ABB RAPID module: Module1.mod

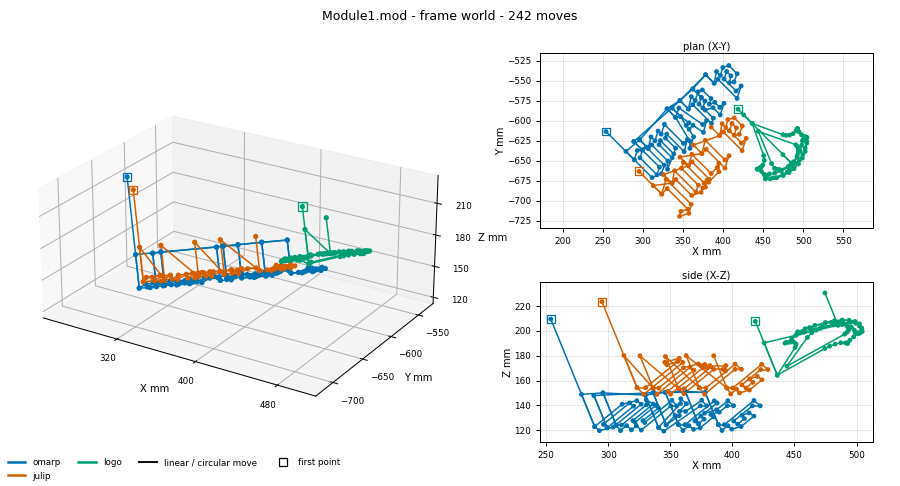
[picture p0: tool path of Module1.mod in frame world, 242 of 244 moves have a stored position in this frame; points joined in program order, loops and branches not executed]
MODULE Module1
    PERS tooldata toolx:=[TRUE,[[148.954,0,67.083],[0.79335334,0,0.608761429,0]],[1,[0,0,1],[1,0,0,0],0,0,0]];
    TASK PERS wobjdata Workobject_2:=[FALSE,TRUE,"",[[233.257625,-636.839625,95.228693814],[0.892399134,-0.099045186,-0.239118017,-0.369643626]],[[0,0,0],[1,0,0,0]]];
    CONST robtarget Target_10:=[[55.302,30.991,100],[0,0,1,0],[-1,1,-2,0],[9E+09,9E+09,9E+09,9E+09,9E+09,9E+09]];
    CONST robtarget Target_20:=[[55.302,30.991,0],[0,0,1,0],[-1,1,-2,0],[9E+09,9E+09,9E+09,9E+09,9E+09,9E+09]];
    CONST robtarget Target_30:=[[91.365,30.991,0],[0,0,1,0],[-1,1,-2,0],[9E+09,9E+09,9E+09,9E+09,9E+09,9E+09]];
    CONST robtarget Target_40:=[[97.105,42.767,0],[0,0,1,0],[-1,1,-2,0],[9E+09,9E+09,9E+09,9E+09,9E+09,9E+09]];
    CONST robtarget Target_50:=[[91.365,52.776,0],[0,0,1,0],[-1,1,-2,0],[9E+09,9E+09,9E+09,9E+09,9E+09,9E+09]];
    CONST robtarget Target_60:=[[54.418,52.776,0],[0,0,1,0],[-1,1,-2,0],[9E+09,9E+09,9E+09,9E+09,9E+09,9E+09]];
    CONST robtarget Target_70:=[[48.825,41.884,0],[0,0,1,0],[-1,1,-2,0],[9E+09,9E+09,9E+09,9E+09,9E+09,9E+09]];
    CONST robtarget Target_80:=[[55.302,30.991,0],[0,0,1,0],[-1,1,-2,0],[9E+09,9E+09,9E+09,9E+09,9E+09,9E+09]];
    CONST robtarget Target_90:=[[55.302,30.991,30],[0,0,1,0],[-1,1,-2,0],[9E+09,9E+09,9E+09,9E+09,9E+09,9E+09]];
    CONST robtarget Target_100:=[[57.714,53.347,30],[0,0,1,0],[-1,1,-2,0],[9E+09,9E+09,9E+09,9E+09,9E+09,9E+09]];
    CONST robtarget Target_110:=[[57.714,53.347,0],[0,0,1,0],[-1,1,-2,0],[9E+09,9E+09,9E+09,9E+09,9E+09,9E+09]];
    CONST robtarget Target_120:=[[57.714,59.499,0],[0,0,1,0],[-1,1,-2,0],[9E+09,9E+09,9E+09,9E+09,9E+09,9E+09]];
    CONST robtarget Target_130:=[[90.706,59.499,0],[0,0,1,0],[-1,1,-2,0],[9E+09,9E+09,9E+09,9E+09,9E+09,9E+09]];
    CONST robtarget Target_140:=[[98.758,51.972,0],[0,0,1,0],[-1,1,-2,0],[9E+09,9E+09,9E+09,9E+09,9E+09,9E+09]];
    CONST robtarget Target_150:=[[91.756,66.151,0],[0,0,1,0],[-1,1,-2,0],[9E+09,9E+09,9E+09,9E+09,9E+09,9E+09]];
    CONST robtarget Target_160:=[[64.974,66.151,0],[0,0,1,0],[-1,1,-2,0],[9E+09,9E+09,9E+09,9E+09,9E+09,9E+09]];
    CONST robtarget Target_170:=[[62.173,71.052,0],[0,0,1,0],[-1,1,-2,0],[9E+09,9E+09,9E+09,9E+09,9E+09,9E+09]];
    CONST robtarget Target_180:=[[89.48,71.052,0],[0,0,1,0],[-1,1,-2,0],[9E+09,9E+09,9E+09,9E+09,9E+09,9E+09]];
    CONST robtarget Target_190:=[[85.36,77.652,0],[0,0,1,0],[-1,1,-2,0],[9E+09,9E+09,9E+09,9E+09,9E+09,9E+09]];
    CONST robtarget Target_200:=[[64.9,77.652,0],[0,0,1,0],[-1,1,-2,0],[9E+09,9E+09,9E+09,9E+09,9E+09,9E+09]];
    CONST robtarget Target_210:=[[61.956,82.215,0],[0,0,1,0],[-1,1,-2,0],[9E+09,9E+09,9E+09,9E+09,9E+09,9E+09]];
    CONST robtarget Target_220:=[[97.748,82.215,0],[0,0,1,0],[-1,1,-2,0],[9E+09,9E+09,9E+09,9E+09,9E+09,9E+09]];
    CONST robtarget Target_230:=[[88.605,95.734,0],[0,0,1,0],[-1,1,-2,0],[9E+09,9E+09,9E+09,9E+09,9E+09,9E+09]];
    CONST robtarget Target_240:=[[88.605,88.907,0],[0,0,1,0],[-1,1,-2,0],[9E+09,9E+09,9E+09,9E+09,9E+09,9E+09]];
    CONST robtarget Target_250:=[[49.745,88.907,0],[0,0,1,0],[-1,1,-2,0],[9E+09,9E+09,9E+09,9E+09,9E+09,9E+09]];
    CONST robtarget Target_260:=[[56.572,77.354,0],[0,0,1,0],[-1,1,-2,0],[9E+09,9E+09,9E+09,9E+09,9E+09,9E+09]];
    CONST robtarget Target_270:=[[50.095,77.354,0],[0,0,1,0],[-1,1,-2,0],[9E+09,9E+09,9E+09,9E+09,9E+09,9E+09]];
    CONST robtarget Target_280:=[[56.922,65.976,0],[0,0,1,0],[-1,1,-2,0],[9E+09,9E+09,9E+09,9E+09,9E+09,9E+09]];
    CONST robtarget Target_290:=[[48.87,65.976,0],[0,0,1,0],[-1,1,-2,0],[9E+09,9E+09,9E+09,9E+09,9E+09,9E+09]];
    CONST robtarget Target_300:=[[57.714,53.347,0],[0,0,1,0],[-1,1,-2,0],[9E+09,9E+09,9E+09,9E+09,9E+09,9E+09]];
    CONST robtarget Target_310:=[[57.714,53.347,30],[0,0,1,0],[-1,1,-2,0],[9E+09,9E+09,9E+09,9E+09,9E+09,9E+09]];
    CONST robtarget Target_320:=[[53.98,104.878,30],[0,0,1,0],[-1,1,-2,0],[9E+09,9E+09,9E+09,9E+09,9E+09,9E+09]];
    CONST robtarget Target_330:=[[53.98,104.878,0],[0,0,1,0],[-1,1,-2,0],[9E+09,9E+09,9E+09,9E+09,9E+09,9E+09]];
    CONST robtarget Target_340:=[[92.492,96.56,0],[0,0,1,0],[-1,1,-2,0],[9E+09,9E+09,9E+09,9E+09,9E+09,9E+09]];
    CONST robtarget Target_350:=[[100.22,90.23,0],[0,0,1,0],[-1,1,-2,0],[9E+09,9E+09,9E+09,9E+09,9E+09,9E+09]];
    CONST robtarget Target_360:=[[92.179,103.629,0],[0,0,1,0],[-1,1,-2,0],[9E+09,9E+09,9E+09,9E+09,9E+09,9E+09]];
    CONST robtarget Target_370:=[[79.793,106.336,0],[0,0,1,0],[-1,1,-2,0],[9E+09,9E+09,9E+09,9E+09,9E+09,9E+09]];
    CONST robtarget Target_380:=[[79.793,113.309,0],[0,0,1,0],[-1,1,-2,0],[9E+09,9E+09,9E+09,9E+09,9E+09,9E+09]];
    CONST robtarget Target_390:=[[97.695,116.224,0],[0,0,1,0],[-1,1,-2,0],[9E+09,9E+09,9E+09,9E+09,9E+09,9E+09]];
    CONST robtarget Target_400:=[[88.848,129.546,0],[0,0,1,0],[-1,1,-2,0],[9E+09,9E+09,9E+09,9E+09,9E+09,9E+09]];
    CONST robtarget Target_410:=[[88.848,122.469,0],[0,0,1,0],[-1,1,-2,0],[9E+09,9E+09,9E+09,9E+09,9E+09,9E+09]];
    CONST robtarget Target_420:=[[47.943,116.119,0],[0,0,1,0],[-1,1,-2,0],[9E+09,9E+09,9E+09,9E+09,9E+09,9E+09]];
    CONST robtarget Target_430:=[[53.98,104.878,0],[0,0,1,0],[-1,1,-2,0],[9E+09,9E+09,9E+09,9E+09,9E+09,9E+09]];
    CONST robtarget Target_440:=[[53.98,104.878,30],[0,0,1,0],[-1,1,-2,0],[9E+09,9E+09,9E+09,9E+09,9E+09,9E+09]];
    CONST robtarget Target_450:=[[58.556,123.595,30],[0,0,1,0],[-1,1,-2,0],[9E+09,9E+09,9E+09,9E+09,9E+09,9E+09]];
    CONST robtarget Target_460:=[[58.556,123.595,0],[0,0,1,0],[-1,1,-2,0],[9E+09,9E+09,9E+09,9E+09,9E+09,9E+09]];
    CONST robtarget Target_470:=[[58.556,131.263,0],[0,0,1,0],[-1,1,-2,0],[9E+09,9E+09,9E+09,9E+09,9E+09,9E+09]];
    CONST robtarget Target_480:=[[96.839,131.263,0],[0,0,1,0],[-1,1,-2,0],[9E+09,9E+09,9E+09,9E+09,9E+09,9E+09]];
    CONST robtarget Target_490:=[[93.38,137.518,0],[0,0,1,0],[-1,1,-2,0],[9E+09,9E+09,9E+09,9E+09,9E+09,9E+09]];
    CONST robtarget Target_500:=[[76.894,137.518,0],[0,0,1,0],[-1,1,-2,0],[9E+09,9E+09,9E+09,9E+09,9E+09,9E+09]];
    CONST robtarget Target_510:=[[82.34,146.497,0],[0,0,1,0],[-1,1,-2,0],[9E+09,9E+09,9E+09,9E+09,9E+09,9E+09]];
    CONST robtarget Target_520:=[[97.06,146.497,0],[0,0,1,0],[-1,1,-2,0],[9E+09,9E+09,9E+09,9E+09,9E+09,9E+09]];
    CONST robtarget Target_530:=[[89.004,160.012,0],[0,0,1,0],[-1,1,-2,0],[9E+09,9E+09,9E+09,9E+09,9E+09,9E+09]];
    CONST robtarget Target_540:=[[89.004,152.806,0],[0,0,1,0],[-1,1,-2,0],[9E+09,9E+09,9E+09,9E+09,9E+09,9E+09]];
    CONST robtarget Target_550:=[[78.627,152.806,0],[0,0,1,0],[-1,1,-2,0],[9E+09,9E+09,9E+09,9E+09,9E+09,9E+09]];
    CONST robtarget Target_560:=[[75.018,146.246,0],[0,0,1,0],[-1,1,-2,0],[9E+09,9E+09,9E+09,9E+09,9E+09,9E+09]];
    CONST robtarget Target_570:=[[71.057,152.806,0],[0,0,1,0],[-1,1,-2,0],[9E+09,9E+09,9E+09,9E+09,9E+09,9E+09]];
    CONST robtarget Target_580:=[[53.357,152.806,0],[0,0,1,0],[-1,1,-2,0],[9E+09,9E+09,9E+09,9E+09,9E+09,9E+09]];
    CONST robtarget Target_590:=[[50.882,147.483,0],[0,0,1,0],[-1,1,-2,0],[9E+09,9E+09,9E+09,9E+09,9E+09,9E+09]];
    CONST robtarget Target_600:=[[56.823,137.086,0],[0,0,1,0],[-1,1,-2,0],[9E+09,9E+09,9E+09,9E+09,9E+09,9E+09]];
    CONST robtarget Target_610:=[[48.901,137.086,0],[0,0,1,0],[-1,1,-2,0],[9E+09,9E+09,9E+09,9E+09,9E+09,9E+09]];
    CONST robtarget Target_620:=[[58.556,123.595,0],[0,0,1,0],[-1,1,-2,0],[9E+09,9E+09,9E+09,9E+09,9E+09,9E+09]];
    CONST robtarget Target_630:=[[58.556,123.595,30],[0,0,1,0],[-1,1,-2,0],[9E+09,9E+09,9E+09,9E+09,9E+09,9E+09]];
    CONST robtarget Target_640:=[[58.524,169.09,30],[0,0,1,0],[-1,1,-2,0],[9E+09,9E+09,9E+09,9E+09,9E+09,9E+09]];
    CONST robtarget Target_650:=[[58.524,169.09,0],[0,0,1,0],[-1,1,-2,0],[9E+09,9E+09,9E+09,9E+09,9E+09,9E+09]];
    CONST robtarget Target_660:=[[58.524,175.96,0],[0,0,1,0],[-1,1,-2,0],[9E+09,9E+09,9E+09,9E+09,9E+09,9E+09]];
    CONST robtarget Target_670:=[[97.451,175.96,0],[0,0,1,0],[-1,1,-2,0],[9E+09,9E+09,9E+09,9E+09,9E+09,9E+09]];
    CONST robtarget Target_680:=[[88.812,190.531,0],[0,0,1,0],[-1,1,-2,0],[9E+09,9E+09,9E+09,9E+09,9E+09,9E+09]];
    CONST robtarget Target_690:=[[88.812,181.58,0],[0,0,1,0],[-1,1,-2,0],[9E+09,9E+09,9E+09,9E+09,9E+09,9E+09]];
    CONST robtarget Target_700:=[[64.353,181.58,0],[0,0,1,0],[-1,1,-2,0],[9E+09,9E+09,9E+09,9E+09,9E+09,9E+09]];
    CONST robtarget Target_710:=[[59.253,190.427,0],[0,0,1,0],[-1,1,-2,0],[9E+09,9E+09,9E+09,9E+09,9E+09,9E+09]];
    CONST robtarget Target_720:=[[68.204,190.427,0],[0,0,1,0],[-1,1,-2,0],[9E+09,9E+09,9E+09,9E+09,9E+09,9E+09]];
    CONST robtarget Target_730:=[[73.512,182.933,0],[0,0,1,0],[-1,1,-2,0],[9E+09,9E+09,9E+09,9E+09,9E+09,9E+09]];
    CONST robtarget Target_740:=[[77.467,187.721,0],[0,0,1,0],[-1,1,-2,0],[9E+09,9E+09,9E+09,9E+09,9E+09,9E+09]];
    CONST robtarget Target_750:=[[72.263,197.713,0],[0,0,1,0],[-1,1,-2,0],[9E+09,9E+09,9E+09,9E+09,9E+09,9E+09]];
    CONST robtarget Target_760:=[[55.506,197.713,0],[0,0,1,0],[-1,1,-2,0],[9E+09,9E+09,9E+09,9E+09,9E+09,9E+09]];
    CONST robtarget Target_770:=[[51.238,190.635,0],[0,0,1,0],[-1,1,-2,0],[9E+09,9E+09,9E+09,9E+09,9E+09,9E+09]];
    CONST robtarget Target_780:=[[56.859,181.476,0],[0,0,1,0],[-1,1,-2,0],[9E+09,9E+09,9E+09,9E+09,9E+09,9E+09]];
    CONST robtarget Target_790:=[[49.053,181.476,0],[0,0,1,0],[-1,1,-2,0],[9E+09,9E+09,9E+09,9E+09,9E+09,9E+09]];
    CONST robtarget Target_800:=[[58.524,169.09,0],[0,0,1,0],[-1,1,-2,0],[9E+09,9E+09,9E+09,9E+09,9E+09,9E+09]];
    CONST robtarget Target_810:=[[58.524,169.09,30],[0,0,1,0],[-1,1,-2,0],[9E+09,9E+09,9E+09,9E+09,9E+09,9E+09]];
    CONST robtarget Target_820:=[[59.96,145.179,30],[0,0,1,0],[-1,1,-2,0],[9E+09,9E+09,9E+09,9E+09,9E+09,9E+09]];
    CONST robtarget Target_830:=[[59.96,145.179,0],[0,0,1,0],[-1,1,-2,0],[9E+09,9E+09,9E+09,9E+09,9E+09,9E+09]];
    CONST robtarget Target_840:=[[64.416,137.257,0],[0,0,1,0],[-1,1,-2,0],[9E+09,9E+09,9E+09,9E+09,9E+09,9E+09]];
    CONST robtarget Target_850:=[[72.461,137.257,0],[0,0,1,0],[-1,1,-2,0],[9E+09,9E+09,9E+09,9E+09,9E+09,9E+09]];
    CONST robtarget Target_860:=[[67.386,145.179,0],[0,0,1,0],[-1,1,-2,0],[9E+09,9E+09,9E+09,9E+09,9E+09,9E+09]];
    CONST robtarget Target_870:=[[59.96,145.179,0],[0,0,1,0],[-1,1,-2,0],[9E+09,9E+09,9E+09,9E+09,9E+09,9E+09]];
    CONST robtarget Target_880:=[[59.96,145.179,30],[0,0,1,0],[-1,1,-2,0],[9E+09,9E+09,9E+09,9E+09,9E+09,9E+09]];
    CONST robtarget Target_890:=[[58.039,110.083,30],[0,0,1,0],[-1,1,-2,0],[9E+09,9E+09,9E+09,9E+09,9E+09,9E+09]];
    CONST robtarget Target_900:=[[58.039,110.083,0],[0,0,1,0],[-1,1,-2,0],[9E+09,9E+09,9E+09,9E+09,9E+09,9E+09]];
    CONST robtarget Target_910:=[[73.132,107.168,0],[0,0,1,0],[-1,1,-2,0],[9E+09,9E+09,9E+09,9E+09,9E+09,9E+09]];
    CONST robtarget Target_920:=[[73.132,111.956,0],[0,0,1,0],[-1,1,-2,0],[9E+09,9E+09,9E+09,9E+09,9E+09,9E+09]];
    CONST robtarget Target_930:=[[58.039,110.083,0],[0,0,1,0],[-1,1,-2,0],[9E+09,9E+09,9E+09,9E+09,9E+09,9E+09]];
    CONST robtarget Target_940:=[[58.039,110.083,30],[0,0,1,0],[-1,1,-2,0],[9E+09,9E+09,9E+09,9E+09,9E+09,9E+09]];
    CONST robtarget Target_950:=[[53.478,46.741,30],[0,0,1,0],[-1,1,-2,0],[9E+09,9E+09,9E+09,9E+09,9E+09,9E+09]];
    CONST robtarget Target_960:=[[53.478,46.741,0],[0,0,1,0],[-1,1,-2,0],[9E+09,9E+09,9E+09,9E+09,9E+09,9E+09]];
    CONST robtarget Target_970:=[[58.982,37.762,0],[0,0,1,0],[-1,1,-2,0],[9E+09,9E+09,9E+09,9E+09,9E+09,9E+09]];
    CONST robtarget Target_980:=[[93.58,37.762,0],[0,0,1,0],[-1,1,-2,0],[9E+09,9E+09,9E+09,9E+09,9E+09,9E+09]];
    CONST robtarget Target_990:=[[88.274,46.741,0],[0,0,1,0],[-1,1,-2,0],[9E+09,9E+09,9E+09,9E+09,9E+09,9E+09]];
    CONST robtarget Target_1000:=[[53.478,46.741,0],[0,0,1,0],[-1,1,-2,0],[9E+09,9E+09,9E+09,9E+09,9E+09,9E+09]];
    CONST robtarget Target_1010:=[[53.478,46.741,30],[0,0,1,0],[-1,1,-2,0],[9E+09,9E+09,9E+09,9E+09,9E+09,9E+09]];
    CONST jointtarget JointTarget_3:=[[0,0,0,0,0,0],[9E+09,9E+09,9E+09,9E+09,9E+09,9E+09]];
    CONST robtarget Target_1020:=[[118.053795712,24.917790512,80],[0,0,1,0],[-1,1,-2,0],[9E+09,9E+09,9E+09,9E+09,9E+09,9E+09]];
    CONST robtarget Target_1030:=[[118.054,24.918,0],[0,0,1,0],[-1,1,-2,0],[9E+09,9E+09,9E+09,9E+09,9E+09,9E+09]];
    CONST robtarget Target_1040:=[[118.054,34.711,0],[0,0,1,0],[-1,1,-2,0],[9E+09,9E+09,9E+09,9E+09,9E+09,9E+09]];
    CONST robtarget Target_1050:=[[160.24,34.711,0],[0,0,1,0],[-1,1,-2,0],[9E+09,9E+09,9E+09,9E+09,9E+09,9E+09]];
    CONST robtarget Target_1060:=[[155.164,26.659,0],[0,0,1,0],[-1,1,-2,0],[9E+09,9E+09,9E+09,9E+09,9E+09,9E+09]];
    CONST robtarget Target_1070:=[[159.015,21.058,0],[0,0,1,0],[-1,1,-2,0],[9E+09,9E+09,9E+09,9E+09,9E+09,9E+09]];
    CONST robtarget Target_1080:=[[165.492,31.911,0],[0,0,1,0],[-1,1,-2,0],[9E+09,9E+09,9E+09,9E+09,9E+09,9E+09]];
    CONST robtarget Target_1090:=[[158.665,41.888,0],[0,0,1,0],[-1,1,-2,0],[9E+09,9E+09,9E+09,9E+09,9E+09,9E+09]];
    CONST robtarget Target_1100:=[[107.376,41.888,0],[0,0,1,0],[-1,1,-2,0],[9E+09,9E+09,9E+09,9E+09,9E+09,9E+09]];
    CONST robtarget Target_1110:=[[118.054,24.918,0],[0,0,1,0],[-1,1,-2,0],[9E+09,9E+09,9E+09,9E+09,9E+09,9E+09]];
    CONST robtarget Target_1120:=[[118.054,24.918,30],[0,0,1,0],[-1,1,-2,0],[9E+09,9E+09,9E+09,9E+09,9E+09,9E+09]];
    CONST robtarget Target_1130:=[[117.489,43.728,0],[0,0,1,0],[-1,1,-2,0],[9E+09,9E+09,9E+09,9E+09,9E+09,9E+09]];
    CONST robtarget Target_1140:=[[117.489,50.177,0],[0,0,1,0],[-1,1,-2,0],[9E+09,9E+09,9E+09,9E+09,9E+09,9E+09]];
    CONST robtarget Target_1150:=[[150.072,50.177,0],[0,0,1,0],[-1,1,-2,0],[9E+09,9E+09,9E+09,9E+09,9E+09,9E+09]];
    CONST robtarget Target_1160:=[[156.421,61.314,0],[0,0,1,0],[-1,1,-2,0],[9E+09,9E+09,9E+09,9E+09,9E+09,9E+09]];
    CONST robtarget Target_1170:=[[153.61,66.726,0],[0,0,1,0],[-1,1,-2,0],[9E+09,9E+09,9E+09,9E+09,9E+09,9E+09]];
    CONST robtarget Target_1180:=[[155.588,69.745,0],[0,0,1,0],[-1,1,-2,0],[9E+09,9E+09,9E+09,9E+09,9E+09,9E+09]];
    CONST robtarget Target_1190:=[[150.072,77.343,0],[0,0,1,0],[-1,1,-2,0],[9E+09,9E+09,9E+09,9E+09,9E+09,9E+09]];
    CONST robtarget Target_1200:=[[150.072,72.176,0],[0,0,1,0],[-1,1,-2,0],[9E+09,9E+09,9E+09,9E+09,9E+09,9E+09]];
    CONST robtarget Target_1210:=[[107.603,72.176,0],[0,0,1,0],[-1,1,-2,0],[9E+09,9E+09,9E+09,9E+09,9E+09,9E+09]];
    CONST robtarget Target_1220:=[[111.979,65.13,0],[0,0,1,0],[-1,1,-2,0],[9E+09,9E+09,9E+09,9E+09,9E+09,9E+09]];
    CONST robtarget Target_1230:=[[146.392,65.13,0],[0,0,1,0],[-1,1,-2,0],[9E+09,9E+09,9E+09,9E+09,9E+09,9E+09]];
    CONST robtarget Target_1240:=[[150.91,56.876,0],[0,0,1,0],[-1,1,-2,0],[9E+09,9E+09,9E+09,9E+09,9E+09,9E+09]];
    CONST robtarget Target_1250:=[[107.381,56.876,0],[0,0,1,0],[-1,1,-2,0],[9E+09,9E+09,9E+09,9E+09,9E+09,9E+09]];
    CONST robtarget Target_1260:=[[117.489,43.728,0],[0,0,1,0],[-1,1,-2,0],[9E+09,9E+09,9E+09,9E+09,9E+09,9E+09]];
    CONST robtarget Target_1270:=[[117.489,43.728,30],[0,0,1,0],[-1,1,-2,0],[9E+09,9E+09,9E+09,9E+09,9E+09,9E+09]];
    CONST robtarget Target_1280:=[[116.365,73.7,0],[0,0,1,0],[-1,1,-2,0],[9E+09,9E+09,9E+09,9E+09,9E+09,9E+09]];
    CONST robtarget Target_1290:=[[116.365,80.093,0],[0,0,1,0],[-1,1,-2,0],[9E+09,9E+09,9E+09,9E+09,9E+09,9E+09]];
    CONST robtarget Target_1300:=[[151.605,80.093,0],[0,0,1,0],[-1,1,-2,0],[9E+09,9E+09,9E+09,9E+09,9E+09,9E+09]];
    CONST robtarget Target_1310:=[[153.709,76.813,0],[0,0,1,0],[-1,1,-2,0],[9E+09,9E+09,9E+09,9E+09,9E+09,9E+09]];
    CONST robtarget Target_1320:=[[153.709,95.194,0],[0,0,1,0],[-1,1,-2,0],[9E+09,9E+09,9E+09,9E+09,9E+09,9E+09]];
    CONST robtarget Target_1330:=[[144.921,102.496,0],[0,0,1,0],[-1,1,-2,0],[9E+09,9E+09,9E+09,9E+09,9E+09,9E+09]];
    CONST robtarget Target_1340:=[[147.621,97.284,0],[0,0,1,0],[-1,1,-2,0],[9E+09,9E+09,9E+09,9E+09,9E+09,9E+09]];
    CONST robtarget Target_1350:=[[147.621,86.727,0],[0,0,1,0],[-1,1,-2,0],[9E+09,9E+09,9E+09,9E+09,9E+09,9E+09]];
    CONST robtarget Target_1360:=[[108.343,86.727,0],[0,0,1,0],[-1,1,-2,0],[9E+09,9E+09,9E+09,9E+09,9E+09,9E+09]];
    CONST robtarget Target_1370:=[[116.365,73.7,0],[0,0,1,0],[-1,1,-2,0],[9E+09,9E+09,9E+09,9E+09,9E+09,9E+09]];
    CONST robtarget Target_1380:=[[116.365,73.7,30],[0,0,1,0],[-1,1,-2,0],[9E+09,9E+09,9E+09,9E+09,9E+09,9E+09]];
    CONST robtarget Target_1390:=[[117.776,96.145,0],[0,0,1,0],[-1,1,-2,0],[9E+09,9E+09,9E+09,9E+09,9E+09,9E+09]];
    CONST robtarget Target_1400:=[[117.776,103.695,0],[0,0,1,0],[-1,1,-2,0],[9E+09,9E+09,9E+09,9E+09,9E+09,9E+09]];
    CONST robtarget Target_1410:=[[156.047,103.695,0],[0,0,1,0],[-1,1,-2,0],[9E+09,9E+09,9E+09,9E+09,9E+09,9E+09]];
    CONST robtarget Target_1420:=[[147.621,118.268,0],[0,0,1,0],[-1,1,-2,0],[9E+09,9E+09,9E+09,9E+09,9E+09,9E+09]];
    CONST robtarget Target_1430:=[[147.621,110.908,0],[0,0,1,0],[-1,1,-2,0],[9E+09,9E+09,9E+09,9E+09,9E+09,9E+09]];
    CONST robtarget Target_1440:=[[107.62,110.908,0],[0,0,1,0],[-1,1,-2,0],[9E+09,9E+09,9E+09,9E+09,9E+09,9E+09]];
    CONST robtarget Target_1450:=[[117.776,96.145,0],[0,0,1,0],[-1,1,-2,0],[9E+09,9E+09,9E+09,9E+09,9E+09,9E+09]];
    CONST robtarget Target_1460:=[[117.776,96.145,30],[0,0,1,0],[-1,1,-2,0],[9E+09,9E+09,9E+09,9E+09,9E+09,9E+09]];
    CONST robtarget Target_1470:=[[117.559,127.676,0],[0,0,1,0],[-1,1,-2,0],[9E+09,9E+09,9E+09,9E+09,9E+09,9E+09]];
    CONST robtarget Target_1480:=[[117.559,134.299,0],[0,0,1,0],[-1,1,-2,0],[9E+09,9E+09,9E+09,9E+09,9E+09,9E+09]];
    CONST robtarget Target_1490:=[[155.683,134.299,0],[0,0,1,0],[-1,1,-2,0],[9E+09,9E+09,9E+09,9E+09,9E+09,9E+09]];
    CONST robtarget Target_1500:=[[147.293,148.725,0],[0,0,1,0],[-1,1,-2,0],[9E+09,9E+09,9E+09,9E+09,9E+09,9E+09]];
    CONST robtarget Target_1510:=[[147.293,140.482,0],[0,0,1,0],[-1,1,-2,0],[9E+09,9E+09,9E+09,9E+09,9E+09,9E+09]];
    CONST robtarget Target_1520:=[[122.564,140.482,0],[0,0,1,0],[-1,1,-2,0],[9E+09,9E+09,9E+09,9E+09,9E+09,9E+09]];
    CONST robtarget Target_1530:=[[117.707,149.313,0],[0,0,1,0],[-1,1,-2,0],[9E+09,9E+09,9E+09,9E+09,9E+09,9E+09]];
    CONST robtarget Target_1540:=[[126.686,149.313,0],[0,0,1,0],[-1,1,-2,0],[9E+09,9E+09,9E+09,9E+09,9E+09,9E+09]];
    CONST robtarget Target_1550:=[[132.132,140.923,0],[0,0,1,0],[-1,1,-2,0],[9E+09,9E+09,9E+09,9E+09,9E+09,9E+09]];
    CONST robtarget Target_1560:=[[136.253,146.222,0],[0,0,1,0],[-1,1,-2,0],[9E+09,9E+09,9E+09,9E+09,9E+09,9E+09]];
    CONST robtarget Target_1570:=[[130.807,156.232,0],[0,0,1,0],[-1,1,-2,0],[9E+09,9E+09,9E+09,9E+09,9E+09,9E+09]];
    CONST robtarget Target_1580:=[[114.321,156.232,0],[0,0,1,0],[-1,1,-2,0],[9E+09,9E+09,9E+09,9E+09,9E+09,9E+09]];
    CONST robtarget Target_1590:=[[109.464,149.019,0],[0,0,1,0],[-1,1,-2,0],[9E+09,9E+09,9E+09,9E+09,9E+09,9E+09]];
    CONST robtarget Target_1600:=[[115.646,140.334,0],[0,0,1,0],[-1,1,-2,0],[9E+09,9E+09,9E+09,9E+09,9E+09,9E+09]];
    CONST robtarget Target_1610:=[[107.992,140.334,0],[0,0,1,0],[-1,1,-2,0],[9E+09,9E+09,9E+09,9E+09,9E+09,9E+09]];
    CONST robtarget Target_1620:=[[117.559,127.676,0],[0,0,1,0],[-1,1,-2,0],[9E+09,9E+09,9E+09,9E+09,9E+09,9E+09]];
    CONST robtarget Target_1630:=[[117.559,127.676,30],[0,0,1,0],[-1,1,-2,0],[9E+09,9E+09,9E+09,9E+09,9E+09,9E+09]];
    CONST robtarget Target_1640:=[[138.252126131,167.190655355,50],[0,0,1,0],[0,-2,1,0],[9E+09,9E+09,9E+09,9E+09,9E+09,9E+09]];
    CONST robtarget Target_1650:=[[138.252126131,167.190655355,0],[0,0,1,0],[-1,-3,2,0],[9E+09,9E+09,9E+09,9E+09,9E+09,9E+09]];
    CONST robtarget Target_1660:=[[182.853126131,148.892655355,0],[0,0,1,0],[-1,-3,2,0],[9E+09,9E+09,9E+09,9E+09,9E+09,9E+09]];
    CONST robtarget Target_1670:=[[188.289126131,145.259655355,0],[0,0,1,0],[-1,-3,2,0],[9E+09,9E+09,9E+09,9E+09,9E+09,9E+09]];
    CONST robtarget Target_1680:=[[191.523126131,139.892655355,0],[0,0,1,0],[-1,-3,2,0],[9E+09,9E+09,9E+09,9E+09,9E+09,9E+09]];
    CONST robtarget Target_1690:=[[191.698126131,137.004655355,0],[0,0,1,0],[-1,-3,2,0],[9E+09,9E+09,9E+09,9E+09,9E+09,9E+09]];
    CONST robtarget Target_1700:=[[191.106126131,134.204655355,0],[0,0,1,0],[-1,-3,2,0],[9E+09,9E+09,9E+09,9E+09,9E+09,9E+09]];
    CONST robtarget Target_1710:=[[189.870126131,131.274655355,0],[0,0,1,0],[-1,-3,2,0],[9E+09,9E+09,9E+09,9E+09,9E+09,9E+09]];
    CONST robtarget Target_1720:=[[190.919126131,131.728655355,0],[0,0,1,0],[-1,-3,2,0],[9E+09,9E+09,9E+09,9E+09,9E+09,9E+09]];
    CONST robtarget Target_1730:=[[196.615126131,133.056655355,0],[0,0,1,0],[-1,-3,2,0],[9E+09,9E+09,9E+09,9E+09,9E+09,9E+09]];
    CONST robtarget Target_1740:=[[202.280126131,132.854655355,0],[0,0,1,0],[-1,-3,2,0],[9E+09,9E+09,9E+09,9E+09,9E+09,9E+09]];
    CONST robtarget Target_1750:=[[204.781126131,132.265655355,0],[0,0,1,0],[-1,-3,2,0],[9E+09,9E+09,9E+09,9E+09,9E+09,9E+09]];
    CONST robtarget Target_1760:=[[206.592126131,131.649655355,0],[0,0,1,0],[-1,-3,2,0],[9E+09,9E+09,9E+09,9E+09,9E+09,9E+09]];
    CONST robtarget Target_1770:=[[206.104126131,134.384655355,0],[0,0,1,0],[-1,-3,2,0],[9E+09,9E+09,9E+09,9E+09,9E+09,9E+09]];
    CONST robtarget Target_1780:=[[207.280126131,137.789655355,0],[0,0,1,0],[-1,-3,2,0],[9E+09,9E+09,9E+09,9E+09,9E+09,9E+09]];
    CONST robtarget Target_1790:=[[211.888126131,143.150655355,0],[0,0,1,0],[-1,-3,2,0],[9E+09,9E+09,9E+09,9E+09,9E+09,9E+09]];
    CONST robtarget Target_1800:=[[216.330126131,150.731655355,-0.07],[0,0,1,0],[-1,-3,2,0],[9E+09,9E+09,9E+09,9E+09,9E+09,9E+09]];
    CONST robtarget Target_1810:=[[219.483126131,160.043655355,0],[0,0,1,0],[-1,-3,2,0],[9E+09,9E+09,9E+09,9E+09,9E+09,9E+09]];
    CONST robtarget Target_1820:=[[219.878126131,163.498655355,0],[0,0,1,0],[-1,-3,2,0],[9E+09,9E+09,9E+09,9E+09,9E+09,9E+09]];
    CONST robtarget Target_1830:=[[219.208126131,161.196655355,0],[0,0,1,0],[-1,-3,2,0],[9E+09,9E+09,9E+09,9E+09,9E+09,9E+09]];
    CONST robtarget Target_1840:=[[213.540126131,150.804655355,0],[0,0,1,0],[-1,-3,2,0],[9E+09,9E+09,9E+09,9E+09,9E+09,9E+09]];
    CONST robtarget Target_1850:=[[210.518126131,148.746655355,0],[0,0,1,0],[-1,-3,2,0],[9E+09,9E+09,9E+09,9E+09,9E+09,9E+09]];
    CONST robtarget Target_1860:=[[206.663126131,147.230655355,0],[0,0,1,0],[-1,-3,2,0],[9E+09,9E+09,9E+09,9E+09,9E+09,9E+09]];
    CONST robtarget Target_1870:=[[199.081126131,148.833655355,0],[0,0,1,0],[-1,-3,2,0],[9E+09,9E+09,9E+09,9E+09,9E+09,9E+09]];
    CONST robtarget Target_1880:=[[152.628126131,165.630655355,0],[0,0,1,0],[-1,-3,2,0],[9E+09,9E+09,9E+09,9E+09,9E+09,9E+09]];
    CONST robtarget Target_1890:=[[204.336126131,186.785655355,0],[0,0,1,0],[-1,-3,2,0],[9E+09,9E+09,9E+09,9E+09,9E+09,9E+09]];
    CONST robtarget Target_1900:=[[207.620126131,186.756655355,0],[0,0,1,0],[-1,-3,2,0],[9E+09,9E+09,9E+09,9E+09,9E+09,9E+09]];
    CONST robtarget Target_1910:=[[211.019126131,185.551655355,0],[0,0,1,0],[-1,-3,2,0],[9E+09,9E+09,9E+09,9E+09,9E+09,9E+09]];
    CONST robtarget Target_1920:=[[214.317126131,182.534655355,0],[0,0,1,0],[-1,-3,2,0],[9E+09,9E+09,9E+09,9E+09,9E+09,9E+09]];
    CONST robtarget Target_1930:=[[216.873126131,178.677655355,0],[0,0,1,0],[-1,-3,2,0],[9E+09,9E+09,9E+09,9E+09,9E+09,9E+09]];
    CONST robtarget Target_1940:=[[219.867126131,170.422655355,0],[0,0,1,0],[-1,-3,2,0],[9E+09,9E+09,9E+09,9E+09,9E+09,9E+09]];
    CONST robtarget Target_1950:=[[218.530126131,176.944655355,0],[0,0,1,0],[-1,-3,2,0],[9E+09,9E+09,9E+09,9E+09,9E+09,9E+09]];
    CONST robtarget Target_1960:=[[215.486126131,184.820655355,0],[0,0,1,0],[-1,-3,2,0],[9E+09,9E+09,9E+09,9E+09,9E+09,9E+09]];
    CONST robtarget Target_1970:=[[210.956126131,191.779655355,0],[0,0,1,0],[-1,-3,2,0],[9E+09,9E+09,9E+09,9E+09,9E+09,9E+09]];
    CONST robtarget Target_1980:=[[207.340126131,196.153655355,0],[0,0,1,0],[-1,-3,2,0],[9E+09,9E+09,9E+09,9E+09,9E+09,9E+09]];
    CONST robtarget Target_1990:=[[206.444126131,198.165655355,0],[0,0,1,0],[-1,-3,2,0],[9E+09,9E+09,9E+09,9E+09,9E+09,9E+09]];
    CONST robtarget Target_2000:=[[206.145126131,200.551655355,0],[0,0,1,0],[-1,-3,2,0],[9E+09,9E+09,9E+09,9E+09,9E+09,9E+09]];
    CONST robtarget Target_2010:=[[206.635126131,202.130655355,0],[0,0,1,0],[-1,-3,2,0],[9E+09,9E+09,9E+09,9E+09,9E+09,9E+09]];
    CONST robtarget Target_2020:=[[206.270126131,202.113655355,0],[0,0,1,0],[-1,-3,2,0],[9E+09,9E+09,9E+09,9E+09,9E+09,9E+09]];
    CONST robtarget Target_2030:=[[205.255126131,201.773655355,0],[0,0,1,0],[-1,-3,2,0],[9E+09,9E+09,9E+09,9E+09,9E+09,9E+09]];
    CONST robtarget Target_2040:=[[200.101126131,200.754655355,0],[0,0,1,0],[-1,-3,2,0],[9E+09,9E+09,9E+09,9E+09,9E+09,9E+09]];
    CONST robtarget Target_2050:=[[194.532126131,201.118655355,0],[0,0,1,0],[-1,-3,2,0],[9E+09,9E+09,9E+09,9E+09,9E+09,9E+09]];
    CONST robtarget Target_2060:=[[189.839126131,202.668655355,0],[0,0,1,0],[-1,-3,2,0],[9E+09,9E+09,9E+09,9E+09,9E+09,9E+09]];
    CONST robtarget Target_2070:=[[189.665126131,202.624655355,0],[0,0,1,0],[-1,-3,2,0],[9E+09,9E+09,9E+09,9E+09,9E+09,9E+09]];
    CONST robtarget Target_2080:=[[189.640126131,202.399655355,0],[0,0,1,0],[-1,-3,2,0],[9E+09,9E+09,9E+09,9E+09,9E+09,9E+09]];
    CONST robtarget Target_2090:=[[190.328126131,199.832655355,0],[0,0,1,0],[-1,-3,2,0],[9E+09,9E+09,9E+09,9E+09,9E+09,9E+09]];
    CONST robtarget Target_2100:=[[190.437126131,194.316655355,0],[0,0,1,0],[-1,-3,2,0],[9E+09,9E+09,9E+09,9E+09,9E+09,9E+09]];
    CONST robtarget Target_2110:=[[188.308126131,189.872655355,0],[0,0,1,0],[-1,-3,2,0],[9E+09,9E+09,9E+09,9E+09,9E+09,9E+09]];
    CONST robtarget Target_2120:=[[184.946126131,186.502655355,0],[0,0,1,0],[-1,-3,2,0],[9E+09,9E+09,9E+09,9E+09,9E+09,9E+09]];
    CONST robtarget Target_2130:=[[181.138126131,184.381655355,0],[0,0,1,0],[-1,-3,2,0],[9E+09,9E+09,9E+09,9E+09,9E+09,9E+09]];
    CONST robtarget Target_2140:=[[138.252126131,167.190655355,0],[0,0,1,0],[-1,-3,2,0],[9E+09,9E+09,9E+09,9E+09,9E+09,9E+09]];
    CONST robtarget Target_2150:=[[138.252126131,167.190655355,30],[0,0,1,0],[-1,-3,2,0],[9E+09,9E+09,9E+09,9E+09,9E+09,9E+09]];
    CONST robtarget Target_2160:=[[218.743126131,166.753655355,0],[0,0,1,0],[-1,-3,2,0],[9E+09,9E+09,9E+09,9E+09,9E+09,9E+09]];
    CONST robtarget Target_2170:=[[221.766126131,164.924655355,0],[0,0,1,0],[-1,-3,2,0],[9E+09,9E+09,9E+09,9E+09,9E+09,9E+09]];
    CONST robtarget Target_2180:=[[222.814126131,163.117655355,0],[0,0,1,0],[-1,-3,2,0],[9E+09,9E+09,9E+09,9E+09,9E+09,9E+09]];
    CONST robtarget Target_2190:=[[223.403126131,160.718655355,0],[0,0,1,0],[-1,-3,2,0],[9E+09,9E+09,9E+09,9E+09,9E+09,9E+09]];
    CONST robtarget Target_2200:=[[223.425126131,155.158655355,0],[0,0,1,0],[-1,-3,2,0],[9E+09,9E+09,9E+09,9E+09,9E+09,9E+09]];
    CONST robtarget Target_2210:=[[221.936126131,149.289655355,0],[0,0,1,0],[-1,-3,2,0],[9E+09,9E+09,9E+09,9E+09,9E+09,9E+09]];
    CONST robtarget Target_2220:=[[214.875126131,137.337655355,0],[0,0,1,0],[-1,-3,2,0],[9E+09,9E+09,9E+09,9E+09,9E+09,9E+09]];
    CONST robtarget Target_2230:=[[208.189126131,129.949655355,0],[0,0,1,0],[-1,-3,2,0],[9E+09,9E+09,9E+09,9E+09,9E+09,9E+09]];
    CONST robtarget Target_2240:=[[213.035126131,134.058655355,0],[0,0,1,0],[-1,-3,2,0],[9E+09,9E+09,9E+09,9E+09,9E+09,9E+09]];
    CONST robtarget Target_2250:=[[218.484126131,140.675655355,0],[0,0,1,0],[-1,-3,2,0],[9E+09,9E+09,9E+09,9E+09,9E+09,9E+09]];
    CONST robtarget Target_2260:=[[223.066126131,148.529655355,0],[0,0,1,0],[-1,-3,2,0],[9E+09,9E+09,9E+09,9E+09,9E+09,9E+09]];
    CONST robtarget Target_2270:=[[225.977126131,156.461655355,0],[0,0,1,0],[-1,-3,2,0],[9E+09,9E+09,9E+09,9E+09,9E+09,9E+09]];
    CONST robtarget Target_2280:=[[227.126126131,164.215655355,0],[0,0,1,0],[-1,-3,2,0],[9E+09,9E+09,9E+09,9E+09,9E+09,9E+09]];
    CONST robtarget Target_2290:=[[226.705126131,172.318655355,0],[0,0,1,0],[-1,-3,2,0],[9E+09,9E+09,9E+09,9E+09,9E+09,9E+09]];
    CONST robtarget Target_2300:=[[224.756126131,180.878655355,0],[0,0,1,0],[-1,-3,2,0],[9E+09,9E+09,9E+09,9E+09,9E+09,9E+09]];
    CONST robtarget Target_2310:=[[220.838126131,189.359655355,0],[0,0,1,0],[-1,-3,2,0],[9E+09,9E+09,9E+09,9E+09,9E+09,9E+09]];
    CONST robtarget Target_2320:=[[214.016126131,197.878655355,0],[0,0,1,0],[-1,-3,2,0],[9E+09,9E+09,9E+09,9E+09,9E+09,9E+09]];
    CONST robtarget Target_2330:=[[208.409126131,203.195655355,0],[0,0,1,0],[-1,-3,2,0],[9E+09,9E+09,9E+09,9E+09,9E+09,9E+09]];
    CONST robtarget Target_2340:=[[211.829126131,199.712655355,0],[0,0,1,0],[-1,-3,2,0],[9E+09,9E+09,9E+09,9E+09,9E+09,9E+09]];
    CONST robtarget Target_2350:=[[217.683126131,191.943655355,0],[0,0,1,0],[-1,-3,2,0],[9E+09,9E+09,9E+09,9E+09,9E+09,9E+09]];
    CONST robtarget Target_2360:=[[221.829126131,184.123655355,0],[0,0,1,0],[-1,-3,2,0],[9E+09,9E+09,9E+09,9E+09,9E+09,9E+09]];
    CONST robtarget Target_2370:=[[223.347126131,176.912655355,0],[0,0,1,0],[-1,-3,2,0],[9E+09,9E+09,9E+09,9E+09,9E+09,9E+09]];
    CONST robtarget Target_2380:=[[222.509126131,169.519655355,0],[0,0,1,0],[-1,-3,2,0],[9E+09,9E+09,9E+09,9E+09,9E+09,9E+09]];
    CONST robtarget Target_2390:=[[221.832126131,168.351655355,0],[0,0,1,0],[-1,-3,2,0],[9E+09,9E+09,9E+09,9E+09,9E+09,9E+09]];
    CONST robtarget Target_2400:=[[220.968126131,167.670655355,0],[0,0,1,0],[-1,-3,2,0],[9E+09,9E+09,9E+09,9E+09,9E+09,9E+09]];
    CONST robtarget Target_2410:=[[218.743126131,166.753655355,0],[0,0,1,0],[-1,-3,2,0],[9E+09,9E+09,9E+09,9E+09,9E+09,9E+09]];
    CONST robtarget Target_2420:=[[218.743126131,166.753655355,30],[0,0,1,0],[-1,-3,2,0],[9E+09,9E+09,9E+09,9E+09,9E+09,9E+09]];
    CONST jointtarget JointTarget_5:=[[0,0,-30,0,-20,0],[9E+09,9E+09,9E+09,9E+09,9E+09,9E+09]];
    PROC omarp()
        MoveJ Target_10,v200,fine,toolx\WObj:=Workobject_2;
        MoveL Target_20,v200,fine,toolx\WObj:=Workobject_2;
        MoveL Target_30,v200,fine,toolx\WObj:=Workobject_2;
        MoveL Target_40,v200,fine,toolx\WObj:=Workobject_2;
        MoveL Target_50,v200,fine,toolx\WObj:=Workobject_2;
        MoveL Target_60,v200,fine,toolx\WObj:=Workobject_2;
        MoveL Target_70,v200,fine,toolx\WObj:=Workobject_2;
        MoveL Target_80,v200,fine,toolx\WObj:=Workobject_2;
        MoveL Target_90,v200,fine,toolx\WObj:=Workobject_2;
        MoveL Target_100,v200,fine,toolx\WObj:=Workobject_2;
        MoveL Target_110,v200,fine,toolx\WObj:=Workobject_2;
        MoveL Target_120,v200,fine,toolx\WObj:=Workobject_2;
        MoveL Target_130,v200,fine,toolx\WObj:=Workobject_2;
        MoveL Target_140,v200,fine,toolx\WObj:=Workobject_2;
        MoveL Target_150,v200,fine,toolx\WObj:=Workobject_2;
        MoveL Target_160,v200,fine,toolx\WObj:=Workobject_2;
        MoveL Target_170,v200,fine,toolx\WObj:=Workobject_2;
        MoveL Target_180,v200,fine,toolx\WObj:=Workobject_2;
        MoveL Target_190,v200,fine,toolx\WObj:=Workobject_2;
        MoveL Target_200,v200,fine,toolx\WObj:=Workobject_2;
        MoveL Target_210,v200,fine,toolx\WObj:=Workobject_2;
        MoveL Target_220,v200,fine,toolx\WObj:=Workobject_2;
        MoveL Target_230,v200,fine,toolx\WObj:=Workobject_2;
        MoveL Target_240,v200,fine,toolx\WObj:=Workobject_2;
        MoveL Target_250,v200,fine,toolx\WObj:=Workobject_2;
        MoveL Target_260,v200,fine,toolx\WObj:=Workobject_2;
        MoveL Target_270,v200,fine,toolx\WObj:=Workobject_2;
        MoveL Target_280,v200,fine,toolx\WObj:=Workobject_2;
        MoveL Target_290,v200,fine,toolx\WObj:=Workobject_2;
        MoveL Target_300,v200,fine,toolx\WObj:=Workobject_2;
        MoveL Target_310,v200,fine,toolx\WObj:=Workobject_2;
        MoveL Target_320,v200,fine,toolx\WObj:=Workobject_2;
        MoveL Target_330,v200,fine,toolx\WObj:=Workobject_2;
        MoveL Target_340,v200,fine,toolx\WObj:=Workobject_2;
        MoveL Target_350,v200,fine,toolx\WObj:=Workobject_2;
        MoveL Target_360,v200,fine,toolx\WObj:=Workobject_2;
        MoveL Target_370,v200,fine,toolx\WObj:=Workobject_2;
        MoveL Target_380,v200,fine,toolx\WObj:=Workobject_2;
        MoveL Target_390,v200,fine,toolx\WObj:=Workobject_2;
        MoveL Target_400,v200,fine,toolx\WObj:=Workobject_2;
        MoveL Target_410,v200,fine,toolx\WObj:=Workobject_2;
        MoveL Target_420,v200,fine,toolx\WObj:=Workobject_2;
        MoveL Target_430,v200,fine,toolx\WObj:=Workobject_2;
        MoveL Target_440,v200,fine,toolx\WObj:=Workobject_2;
        MoveL Target_450,v200,fine,toolx\WObj:=Workobject_2;
        MoveL Target_460,v200,fine,toolx\WObj:=Workobject_2;
        MoveL Target_470,v200,fine,toolx\WObj:=Workobject_2;
        MoveL Target_480,v200,fine,toolx\WObj:=Workobject_2;
        MoveL Target_490,v200,fine,toolx\WObj:=Workobject_2;
        MoveL Target_500,v200,fine,toolx\WObj:=Workobject_2;
        MoveL Target_510,v200,fine,toolx\WObj:=Workobject_2;
        MoveL Target_520,v200,fine,toolx\WObj:=Workobject_2;
        MoveL Target_530,v200,fine,toolx\WObj:=Workobject_2;
        MoveL Target_540,v200,fine,toolx\WObj:=Workobject_2;
        MoveL Target_550,v200,fine,toolx\WObj:=Workobject_2;
        MoveL Target_560,v200,fine,toolx\WObj:=Workobject_2;
        MoveL Target_570,v200,fine,toolx\WObj:=Workobject_2;
        MoveL Target_580,v200,fine,toolx\WObj:=Workobject_2;
        MoveL Target_590,v200,fine,toolx\WObj:=Workobject_2;
        MoveL Target_600,v200,fine,toolx\WObj:=Workobject_2;
        MoveL Target_610,v200,fine,toolx\WObj:=Workobject_2;
        MoveL Target_620,v200,fine,toolx\WObj:=Workobject_2;
        MoveL Target_630,v200,fine,toolx\WObj:=Workobject_2;
        MoveL Target_640,v200,fine,toolx\WObj:=Workobject_2;
        MoveL Target_650,v200,fine,toolx\WObj:=Workobject_2;
        MoveL Target_660,v200,fine,toolx\WObj:=Workobject_2;
        MoveL Target_670,v200,fine,toolx\WObj:=Workobject_2;
        MoveL Target_680,v200,fine,toolx\WObj:=Workobject_2;
        MoveL Target_690,v200,fine,toolx\WObj:=Workobject_2;
        MoveL Target_700,v200,fine,toolx\WObj:=Workobject_2;
        MoveL Target_710,v200,fine,toolx\WObj:=Workobject_2;
        MoveL Target_720,v200,fine,toolx\WObj:=Workobject_2;
        MoveL Target_730,v200,fine,toolx\WObj:=Workobject_2;
        MoveL Target_740,v200,fine,toolx\WObj:=Workobject_2;
        MoveL Target_750,v200,fine,toolx\WObj:=Workobject_2;
        MoveL Target_760,v200,fine,toolx\WObj:=Workobject_2;
        MoveL Target_770,v200,fine,toolx\WObj:=Workobject_2;
        MoveL Target_780,v200,fine,toolx\WObj:=Workobject_2;
        MoveL Target_790,v200,fine,toolx\WObj:=Workobject_2;
        MoveL Target_800,v200,fine,toolx\WObj:=Workobject_2;
        MoveL Target_810,v200,fine,toolx\WObj:=Workobject_2;
        MoveL Target_820,v200,fine,toolx\WObj:=Workobject_2;
        MoveL Target_830,v200,fine,toolx\WObj:=Workobject_2;
        MoveL Target_840,v200,fine,toolx\WObj:=Workobject_2;
        MoveL Target_850,v200,fine,toolx\WObj:=Workobject_2;
        MoveL Target_860,v200,fine,toolx\WObj:=Workobject_2;
        MoveL Target_870,v200,fine,toolx\WObj:=Workobject_2;
        MoveL Target_880,v200,fine,toolx\WObj:=Workobject_2;
        MoveL Target_890,v200,fine,toolx\WObj:=Workobject_2;
        MoveL Target_900,v200,fine,toolx\WObj:=Workobject_2;
        MoveL Target_910,v200,fine,toolx\WObj:=Workobject_2;
        MoveL Target_920,v200,fine,toolx\WObj:=Workobject_2;
        MoveL Target_930,v200,fine,toolx\WObj:=Workobject_2;
        MoveL Target_940,v200,fine,toolx\WObj:=Workobject_2;
        MoveL Target_950,v200,fine,toolx\WObj:=Workobject_2;
        MoveL Target_960,v200,fine,toolx\WObj:=Workobject_2;
        MoveL Target_970,v200,fine,toolx\WObj:=Workobject_2;
        MoveL Target_980,v200,fine,toolx\WObj:=Workobject_2;
        MoveL Target_990,v200,fine,toolx\WObj:=Workobject_2;
        MoveL Target_1000,v200,fine,toolx\WObj:=Workobject_2;
        MoveL Target_1010,v200,fine,toolx\WObj:=Workobject_2;
    ENDPROC
    PROC goHome()
        MoveAbsJ JointTarget_3,v200,z10,toolx\WObj:=Workobject_2;
    ENDPROC
    PROC julip()
        MoveJ Target_1020,v200,fine,toolx\WObj:=Workobject_2;
        MoveL Target_1030,v200,fine,toolx\WObj:=Workobject_2;
        MoveL Target_1040,v200,fine,toolx\WObj:=Workobject_2;
        MoveL Target_1050,v200,fine,toolx\WObj:=Workobject_2;
        MoveL Target_1060,v200,fine,toolx\WObj:=Workobject_2;
        MoveL Target_1070,v200,fine,toolx\WObj:=Workobject_2;
        MoveL Target_1080,v200,fine,toolx\WObj:=Workobject_2;
        MoveL Target_1090,v200,fine,toolx\WObj:=Workobject_2;
        MoveL Target_1100,v200,fine,toolx\WObj:=Workobject_2;
        MoveL Target_1110,v200,fine,toolx\WObj:=Workobject_2;
        MoveL Target_1120,v200,fine,toolx\WObj:=Workobject_2;
        MoveL Target_1130,v200,fine,toolx\WObj:=Workobject_2;
        MoveL Target_1140,v200,fine,toolx\WObj:=Workobject_2;
        MoveL Target_1150,v200,fine,toolx\WObj:=Workobject_2;
        MoveL Target_1160,v200,fine,toolx\WObj:=Workobject_2;
        MoveL Target_1170,v200,fine,toolx\WObj:=Workobject_2;
        MoveL Target_1180,v200,fine,toolx\WObj:=Workobject_2;
        MoveL Target_1190,v200,fine,toolx\WObj:=Workobject_2;
        MoveL Target_1200,v200,fine,toolx\WObj:=Workobject_2;
        MoveL Target_1210,v200,fine,toolx\WObj:=Workobject_2;
        MoveL Target_1220,v200,fine,toolx\WObj:=Workobject_2;
        MoveL Target_1230,v200,fine,toolx\WObj:=Workobject_2;
        MoveL Target_1240,v200,fine,toolx\WObj:=Workobject_2;
        MoveL Target_1250,v200,fine,toolx\WObj:=Workobject_2;
        MoveL Target_1260,v200,fine,toolx\WObj:=Workobject_2;
        MoveL Target_1270,v200,fine,toolx\WObj:=Workobject_2;
        MoveL Target_1280,v200,fine,toolx\WObj:=Workobject_2;
        MoveL Target_1290,v200,fine,toolx\WObj:=Workobject_2;
        MoveL Target_1300,v200,fine,toolx\WObj:=Workobject_2;
        MoveL Target_1310,v200,fine,toolx\WObj:=Workobject_2;
        MoveL Target_1320,v200,fine,toolx\WObj:=Workobject_2;
        MoveL Target_1330,v200,fine,toolx\WObj:=Workobject_2;
        MoveL Target_1340,v200,fine,toolx\WObj:=Workobject_2;
        MoveL Target_1350,v200,fine,toolx\WObj:=Workobject_2;
        MoveL Target_1360,v200,fine,toolx\WObj:=Workobject_2;
        MoveL Target_1370,v200,fine,toolx\WObj:=Workobject_2;
        MoveL Target_1380,v200,fine,toolx\WObj:=Workobject_2;
        MoveL Target_1390,v200,fine,toolx\WObj:=Workobject_2;
        MoveL Target_1400,v200,fine,toolx\WObj:=Workobject_2;
        MoveL Target_1410,v200,fine,toolx\WObj:=Workobject_2;
        MoveL Target_1420,v200,fine,toolx\WObj:=Workobject_2;
        MoveL Target_1430,v200,fine,toolx\WObj:=Workobject_2;
        MoveL Target_1440,v200,fine,toolx\WObj:=Workobject_2;
        MoveL Target_1450,v200,fine,toolx\WObj:=Workobject_2;
        MoveL Target_1460,v200,fine,toolx\WObj:=Workobject_2;
        MoveL Target_1470,v200,fine,toolx\WObj:=Workobject_2;
        MoveL Target_1480,v200,fine,toolx\WObj:=Workobject_2;
        MoveL Target_1490,v200,fine,toolx\WObj:=Workobject_2;
        MoveL Target_1500,v200,fine,toolx\WObj:=Workobject_2;
        MoveL Target_1510,v200,fine,toolx\WObj:=Workobject_2;
        MoveL Target_1520,v200,fine,toolx\WObj:=Workobject_2;
        MoveL Target_1530,v200,fine,toolx\WObj:=Workobject_2;
        MoveL Target_1540,v200,fine,toolx\WObj:=Workobject_2;
        MoveL Target_1550,v200,fine,toolx\WObj:=Workobject_2;
        MoveL Target_1560,v200,fine,toolx\WObj:=Workobject_2;
        MoveL Target_1570,v200,fine,toolx\WObj:=Workobject_2;
        MoveL Target_1580,v200,fine,toolx\WObj:=Workobject_2;
        MoveL Target_1590,v200,fine,toolx\WObj:=Workobject_2;
        MoveL Target_1600,v200,fine,toolx\WObj:=Workobject_2;
        MoveL Target_1610,v200,fine,toolx\WObj:=Workobject_2;
        MoveL Target_1620,v200,fine,toolx\WObj:=Workobject_2;
        MoveL Target_1630,v200,fine,toolx\WObj:=Workobject_2;
    ENDPROC
    PROC logo()
        MoveJ Target_1640,v1000,z100,toolx\WObj:=Workobject_2;
        MoveL Target_1650,v200,fine,toolx\WObj:=Workobject_2;
        MoveL Target_1660,v200,fine,toolx\WObj:=Workobject_2;
        MoveL Target_1670,v200,z10,toolx\WObj:=Workobject_2;
        MoveL Target_1680,v200,z10,toolx\WObj:=Workobject_2;
        MoveL Target_1690,v200,z10,toolx\WObj:=Workobject_2;
        MoveL Target_1700,v200,z10,toolx\WObj:=Workobject_2;
        MoveL Target_1710,v200,fine,toolx\WObj:=Workobject_2;
        MoveL Target_1720,v200,z10,toolx\WObj:=Workobject_2;
        MoveL Target_1730,v200,z10,toolx\WObj:=Workobject_2;
        MoveL Target_1740,v200,z10,toolx\WObj:=Workobject_2;
        MoveL Target_1750,v200,z10,toolx\WObj:=Workobject_2;
        MoveL Target_1760,v200,fine,toolx\WObj:=Workobject_2;
        MoveL Target_1770,v200,z10,toolx\WObj:=Workobject_2;
        MoveL Target_1780,v200,z10,toolx\WObj:=Workobject_2;
        MoveL Target_1790,v200,z10,toolx\WObj:=Workobject_2;
        MoveL Target_1800,v200,z10,toolx\WObj:=Workobject_2;
        MoveL Target_1810,v200,z10,toolx\WObj:=Workobject_2;
        MoveL Target_1820,v200,fine,toolx\WObj:=Workobject_2;
        MoveL Target_1830,v200,z10,toolx\WObj:=Workobject_2;
        MoveL Target_1840,v200,z10,toolx\WObj:=Workobject_2;
        MoveL Target_1850,v200,z10,toolx\WObj:=Workobject_2;
        MoveL Target_1860,v200,z10,toolx\WObj:=Workobject_2;
        MoveL Target_1870,v200,z10,toolx\WObj:=Workobject_2;
        MoveL Target_1880,v200,fine,toolx\WObj:=Workobject_2;
        MoveL Target_1890,v200,z10,toolx\WObj:=Workobject_2;
        MoveL Target_1900,v200,z10,toolx\WObj:=Workobject_2;
        MoveL Target_1910,v200,z10,toolx\WObj:=Workobject_2;
        MoveL Target_1920,v200,z10,toolx\WObj:=Workobject_2;
        MoveL Target_1930,v200,z10,toolx\WObj:=Workobject_2;
        MoveL Target_1940,v200,fine,toolx\WObj:=Workobject_2;
        MoveL Target_1950,v200,z10,toolx\WObj:=Workobject_2;
        MoveL Target_1960,v200,z10,toolx\WObj:=Workobject_2;
        MoveL Target_1970,v200,z10,toolx\WObj:=Workobject_2;
        MoveL Target_1980,v200,z10,toolx\WObj:=Workobject_2;
        MoveL Target_1990,v200,z10,toolx\WObj:=Workobject_2;
        MoveL Target_2000,v200,z10,toolx\WObj:=Workobject_2;
        MoveL Target_2010,v200,fine,toolx\WObj:=Workobject_2;
        MoveL Target_2020,v200,z10,toolx\WObj:=Workobject_2;
        MoveL Target_2030,v200,z10,toolx\WObj:=Workobject_2;
        MoveL Target_2040,v200,z10,toolx\WObj:=Workobject_2;
        MoveL Target_2050,v200,z10,toolx\WObj:=Workobject_2;
        MoveL Target_2060,v200,z10,toolx\WObj:=Workobject_2;
        MoveL Target_2070,v200,z10,toolx\WObj:=Workobject_2;
        MoveL Target_2080,v200,z10,toolx\WObj:=Workobject_2;
        MoveL Target_2090,v200,z10,toolx\WObj:=Workobject_2;
        MoveL Target_2100,v200,z10,toolx\WObj:=Workobject_2;
        MoveL Target_2110,v200,z10,toolx\WObj:=Workobject_2;
        MoveL Target_2120,v200,z10,toolx\WObj:=Workobject_2;
        MoveL Target_2130,v200,z10,toolx\WObj:=Workobject_2;
        MoveL Target_2140,v200,fine,toolx\WObj:=Workobject_2;
        MoveL Target_2150,v200,z10,toolx\WObj:=Workobject_2;
        MoveL Target_2160,v200,fine,toolx\WObj:=Workobject_2;
        MoveL Target_2170,v200,z10,toolx\WObj:=Workobject_2;
        MoveL Target_2180,v200,z10,toolx\WObj:=Workobject_2;
        MoveL Target_2190,v200,z10,toolx\WObj:=Workobject_2;
        MoveL Target_2200,v200,z10,toolx\WObj:=Workobject_2;
        MoveL Target_2210,v200,z10,toolx\WObj:=Workobject_2;
        MoveL Target_2220,v200,z10,toolx\WObj:=Workobject_2;
        MoveL Target_2230,v200,fine,toolx\WObj:=Workobject_2;
        MoveL Target_2240,v200,z10,toolx\WObj:=Workobject_2;
        MoveL Target_2250,v200,z10,toolx\WObj:=Workobject_2;
        MoveL Target_2260,v200,z10,toolx\WObj:=Workobject_2;
        MoveL Target_2270,v200,z10,toolx\WObj:=Workobject_2;
        MoveL Target_2280,v200,z10,toolx\WObj:=Workobject_2;
        MoveL Target_2290,v200,z10,toolx\WObj:=Workobject_2;
        MoveL Target_2300,v200,z10,toolx\WObj:=Workobject_2;
        MoveL Target_2310,v200,z10,toolx\WObj:=Workobject_2;
        MoveL Target_2320,v200,z10,toolx\WObj:=Workobject_2;
        MoveL Target_2330,v200,fine,toolx\WObj:=Workobject_2;
        MoveL Target_2340,v200,z10,toolx\WObj:=Workobject_2;
        MoveL Target_2350,v200,z10,toolx\WObj:=Workobject_2;
        MoveL Target_2360,v200,z10,toolx\WObj:=Workobject_2;
        MoveL Target_2370,v200,z10,toolx\WObj:=Workobject_2;
        MoveL Target_2380,v200,z10,toolx\WObj:=Workobject_2;
        MoveL Target_2390,v200,z10,toolx\WObj:=Workobject_2;
        MoveL Target_2400,v200,z10,toolx\WObj:=Workobject_2;
        MoveL Target_2410,v200,fine,toolx\WObj:=Workobject_2;
        MoveL Target_2420,v200,z10,toolx\WObj:=Workobject_2;
    ENDPROC
    PROC mantenimiento()
        MoveAbsJ JointTarget_5,v200,z10,toolx\WObj:=Workobject_2;
    ENDPROC
    PROC main()
        Reset DO_01;
        Reset DO_02;
        goHome;
        WHILE TRUE DO
        IF DI_01=1 THEN
        Set DO_01;
        omarp;
        julip;
        logo;
        goHome;
        Reset DO_01;
        ENDIF

        IF DI_02=1 THEN
         Set DO_02;
        mantenimiento;
        WaitDI DI_02,1;
        goHome;
        Reset DO_02;
        ENDIF

        ENDWHILE



    ENDPROC
ENDMODULE
